{attribute addProperty BoxType "KL2819"}
{attribute addProperty Id "Channel_1Channel_796AE09F00"}
{attribute addProperty CRC "2203114728"}
{attribute addProperty SizeInBites "0"}
{attribute addProperty SizeInBytes "0"}
TYPE KL2819_8350DCE8 :
STRUCT
	{attribute addProperty Name "Channel_1"}
	Channel_1 : Channel_796AE09F;
END_STRUCT
END_TYPE

(* stored: Version 1.2.0.0, ProductVersion 3.1.4024.9
   DUT KL2819_8350DCE8: Id {57f2aa19-4b45-42d1-a6b0-7ad86e08080f} *)
